Universal Robots PolyScope program: punto1_iniciales.urp

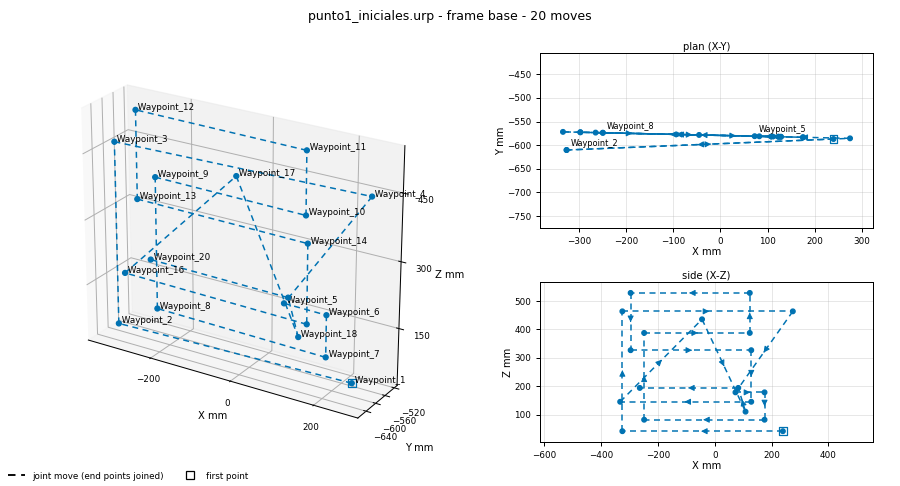
[picture p0: tool path of punto1_iniciales.urp in frame base, 20 of 20 moves have a stored position in this frame; points joined in program order, loops and branches not executed]
Program punto1_iniciales (installation=default directory=/ursim/programs createdIn=3.15.8.106339 lastSavedIn=3.15.8.106339 robotSerialNumber=2018359999)
Calibrated DH parameters: a=[0, -0.425, -0.39225, 0, 0, 0]; d=[0.089159, 0, 0, 0.10915, 0.09465, 0.0823]; alpha=[1.570796, 0, 0, 1.570796, -1.570796, 0]; deltaTheta=[0, 0, 0, 0, 0, 0]
Robot Program (runOnlyOnce=false)
  Popup Message (haltProgram=false message=se va a realizar la c inputType=Text)
  MoveJ speed 60 deg/s, acceleration 80 deg/s^2 (useActiveTCP=true)
    Waypoint Waypoint_1: TCP in base x=239.371 y=-586.942 z=41.673 mm, rx=-0.0012 ry=3.1163 rz=0.0389 rad; joints [-58.158, -129.422, -98.861, -42.175, 91.975, 31.79] deg
    Wait Sleep waitTime=0.5
    Waypoint Waypoint_2: TCP in base x=-325.803 y=-610.224 z=41.673 mm, rx=-0.0012 ry=3.1163 rz=0.0389 rad; joints [-109.127, -134.954, -87.149, -49.719, 90.888, -19.186] deg
    Wait Sleep waitTime=0.5
    Waypoint Waypoint_3: TCP in base x=-325.803 y=-610.224 z=463.672 mm, rx=-0.0012 ry=3.1163 rz=0.0389 rad; joints [-109.127, -119.537, -47.198, -105.088, 90.888, -19.186] deg
    Wait Sleep waitTime=0.5
    Waypoint Waypoint_4: TCP in base x=274.385 y=-585.5 z=463.672 mm, rx=-0.0012 ry=3.1163 rz=0.0389 rad; joints [-55.43, -111.591, -59.287, -99.485, 91.994, 34.519] deg
  Popup Message (haltProgram=false message=se va a realizar la g inputType=Text)
  MoveJ speed 60 deg/s, acceleration 80 deg/s^2 (useActiveTCP=true)
    Waypoint Waypoint_5: TCP in base x=72.438 y=-580.945 z=178.47 mm, rx=-0.0012 ry=3.1163 rz=0.0389 rad; joints [-72.405, -111.893, -102.445, -56.592, 91.801, 17.535] deg
    Wait Sleep waitTime=0.5
    Waypoint Waypoint_6: TCP in base x=174.81 y=-583.254 z=178.47 mm, rx=-0.0012 ry=3.1163 rz=0.0389 rad; joints [-63.253, -114.602, -98.43, -57.6, 91.926, 26.691] deg
    Wait Sleep waitTime=0.5
    Waypoint Waypoint_7: TCP in base x=174.81 y=-583.254 z=82.07 mm, rx=-0.0012 ry=3.1163 rz=0.0389 rad; joints [-63.253, -122.985, -102.623, -45.023, 91.926, 26.691] deg
    Wait Sleep waitTime=0.5
    Waypoint Waypoint_8: TCP in base x=-249.081 y=-573.694 z=82.07 mm, rx=-0.0012 ry=3.1163 rz=0.0389 rad; joints [-103.56, -124.585, -99.294, -47.848, 91.06, -13.621] deg
    Wait Sleep waitTime=0.5
    Waypoint Waypoint_9: TCP in base x=-249.081 y=-573.694 z=387.669 mm, rx=-0.0012 ry=3.1163 rz=0.0389 rad; joints [-103.56, -108.13, -74.834, -88.763, 91.06, -13.621] deg
    Wait Sleep waitTime=0.5
    Waypoint Waypoint_10: TCP in base x=122.823 y=-582.082 z=387.668 mm, rx=-0.0012 ry=3.1163 rz=0.0389 rad; joints [-67.776, -103.712, -80.798, -86.272, 91.87, 22.167] deg
  Popup Message (haltProgram=false message=se realiza la s inputType=Text)
  MoveJ speed 60 deg/s, acceleration 80 deg/s^2 (useActiveTCP=true)
    Waypoint Waypoint_11: TCP in base x=122.823 y=-582.082 z=528.465 mm, rx=-0.0012 ry=3.1163 rz=0.0389 rad; joints [-67.776, -105.909, -57.177, -107.696, 91.87, 22.167] deg
    Wait Sleep waitTime=0.5
    Waypoint Waypoint_12: TCP in base x=-296.669 y=-572.621 z=528.465 mm, rx=-0.0012 ry=3.1163 rz=0.0389 rad; joints [-107.765, -114.557, -44.849, -112.395, 90.931, -17.824] deg
    Wait Sleep waitTime=0.5
    Waypoint Waypoint_13: TCP in base x=-296.669 y=-572.621 z=326.867 mm, rx=-0.0012 ry=3.1163 rz=0.0389 rad; joints [-107.765, -111.846, -78.664, -81.29, 90.931, -17.824] deg
    Wait Sleep waitTime=0.5
    Waypoint Waypoint_14: TCP in base x=128.022 y=-582.199 z=326.867 mm, rx=-0.0012 ry=3.1163 rz=0.0389 rad; joints [-67.311, -105.136, -87.983, -77.647, 91.877, 22.631] deg
    Wait Sleep waitTime=0.5
    Waypoint Waypoint_15: TCP in base x=128.022 y=-582.199 z=145.268 mm, rx=-0.0012 ry=3.1163 rz=0.0389 rad; joints [-67.311, -115.812, -102.464, -52.491, 91.877, 22.631] deg
    Wait Sleep waitTime=0.5
    Waypoint Waypoint_16: TCP in base x=-333.459 y=-571.791 z=145.269 mm, rx=-0.0012 ry=3.1163 rz=0.0389 rad; joints [-110.864, -123.178, -89.938, -58.732, 90.832, -20.922] deg
  Popup Message (haltProgram=false message=se realiza la a inputType=Text)
  MoveJ speed 60 deg/s, acceleration 80 deg/s^2 (useActiveTCP=true)
    Waypoint Waypoint_17: TCP in base x=-45.246 y=-578.291 z=435.667 mm, rx=-0.0012 ry=3.1163 rz=0.0389 rad; joints [-83.856, -101.584, -76.296, -93.389, 91.581, 6.082] deg
    Wait Sleep waitTime=0.5
    Waypoint Waypoint_18: TCP in base x=107.914 y=-581.745 z=110.469 mm, rx=-0.0012 ry=3.1163 rz=0.0389 rad; joints [-69.122, -118.488, -104.733, -47.604, 91.852, 20.82] deg
    Wait Sleep waitTime=0.5
    Waypoint Waypoint_19: TCP in base x=82.322 y=-581.168 z=194.067 mm, rx=-0.0012 ry=3.1163 rz=0.0389 rad; joints [-71.48, -110.894, -101.201, -58.806, 91.816, 18.461] deg
    Wait Sleep waitTime=0.5
    Waypoint Waypoint_20: TCP in base x=-264.388 y=-573.349 z=194.067 mm, rx=-0.0012 ry=3.1163 rz=0.0389 rad; joints [-104.935, -116.193, -92.997, -62.562, 91.019, -14.996] deg
